PROGRAM Process
VAR
	fbAGV: AGV;
END_VAR

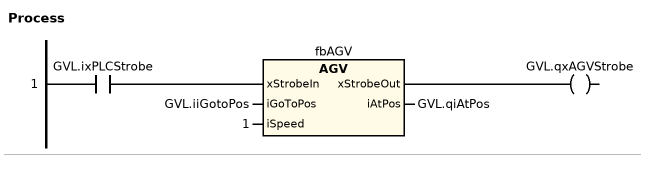
// NETWORK 1
fbAGV(xStrobeIn := GVL.ixPLCStrobe, iGoToPos := GVL.iiGotoPos, iSpeed := 1, iAtPos => GVL.qiAtPos); // AGV
GVL.qxAGVStrobe := fbAGV.xStrobeOut;

END_PROGRAM

(* stored: Version 1.1.0.1, ProductVersion 3.1.4022.12
   POU Process: Id {6818f4c5-9d6b-409a-beb2-84729a516a70}, SpecialFunc None *)
